{attribute 'linkalways'} 
{attribute 'no_explicit_call' := 'This FB is a CLASS and must be accessed using methods or properties'}
{attribute 'enable_dynamic_creation'}
FUNCTION_BLOCK FINAL SIN_LREAL EXTENDS Node
VAR
	in : _LREAL(0.0);
	out : _LREAL(0.0);
END_VAR

METHOD PUBLIC Clone : I_Node
VAR
	pNode : POINTER TO SIN_LREAL;
END_VAR
pNode := __NEW(SIN_LREAL);
Clone := pNode^;
END_METHOD

METHOD FB_init : BOOL
VAR_INPUT
	bInitRetains : BOOL; // if TRUE, the retain variables are initialized (warm start / cold start)
	bInCopyCode : BOOL;  // if TRUE, the instance afterwards gets moved into the copy code (online change)
END_VAR
AddInput('in',THIS^.in);
AddOutput('out', THIS^.out);
END_METHOD

METHOD PROTECTED OnExecute
VAR
END_VAR
out.Value := SIN(in.Value);
END_METHOD

END_FUNCTION_BLOCK

(* stored: Version 1.1.0.1, ProductVersion 3.1.4024.15
   POU SIN_LREAL: Id {7da33879-da26-4559-bbf5-8ba33e91ea11}, SpecialFunc None
   Folder Constructor: Id {beb37dbf-b9ea-4b90-b7da-4ab23800a4af}
   Method Clone: Id {3f2c9df8-0e78-48ea-b7a1-2f02531e4393}
   Method FB_init: Id {4f2f3203-6fc1-4b88-bce4-4a038fb266ea}
   Method OnExecute: Id {736cdd4b-d79a-472b-98a1-1dda2e2e288a} *)
